PROGRAM POU_TempControl
VAR
END_VAR

GVL_IO.lrExtruderTemp := GVL_IO.lrRawTemp/10.0;

END_PROGRAM

(* stored: Version 1.1.0.1, ProductVersion 3.1.4024.2
   POU POU_TempControl: Id {06724fef-7179-4225-9eab-b990c6f641a1}, SpecialFunc None *)
